% RSLogix 500 project 04_P9_ASHLEY_J.RSS, saved by version 8.30.00.16 %
PROJECT "UNTITLED"    % processor: Bul.1763 MicroLogix 1100 Series B %

PROGRAM FILES
  LAD 2 "MAIN"  3 rungs
  LAD 3 "MODE_CTRLS"  13 rungs
  LAD 4 "DATA_CTRL"  9 rungs

DATA FILES
  O0 OUTPUT  4 elements
  I1 INPUT  6 elements
  S2 STATUS  66 elements
  B3 BINARY  10 elements
  T4 TIMER  4 elements
  C5 COUNTER  1 elements
  R6 CONTROL  1 elements
  N7 INTEGER  4 elements
  F8 FLOAT  1 elements
  ST9 STRINGS  10 elements

LADDER 2 "MAIN"
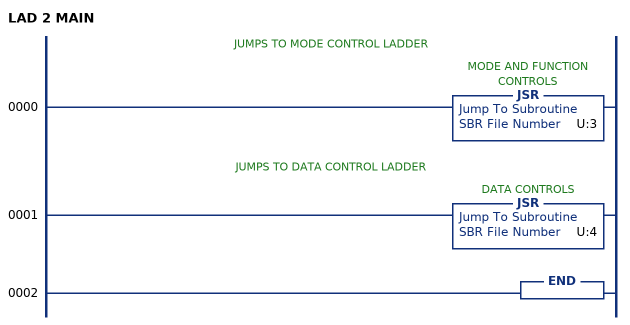
% Rung: 0 %
% JUMPS TO MODE CONTROL LADDER %
SOR JSR U:3 EOR
%   U:3  "MODE AND FUNCTION CONTROLS" %
% Rung: 1 %
% JUMPS TO DATA CONTROL LADDER %
SOR JSR U:4 EOR
%   U:4  "DATA CONTROLS" %
% Rung: 2 %
SOR END EOR

LADDER 3 "MODE_CTRLS"
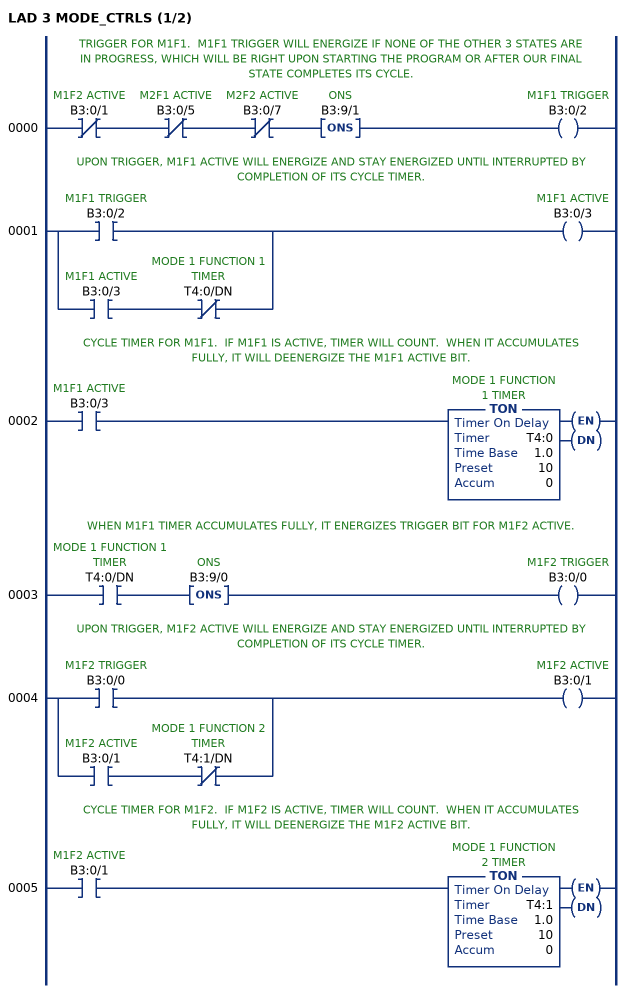
% Rung: 0 %
% TRIGGER FOR M1F1.  M1F1 TRIGGER WILL ENERGIZE IF NONE OF THE OTHER 3 STATES ARE IN PROGRESS, WHICH WILL BE RIGHT UPON STARTING THE PROGRAM OR AFTER OUR FINAL STATE COMPLETES ITS CYCLE. %
SOR XIO B3:0/1 XIO B3:0/5 XIO B3:0/7 ONS B3:9/1 OTE B3:0/2 EOR
%   B3:0/1  "M1F2 ACTIVE" %
%   B3:0/5  "M2F1 ACTIVE" %
%   B3:0/7  "M2F2 ACTIVE" %
%   B3:9/1  "ONS" %
%   B3:0/2  "M1F1 TRIGGER" %
% Rung: 1 %
% UPON TRIGGER, M1F1 ACTIVE WILL ENERGIZE AND STAY ENERGIZED UNTIL INTERRUPTED BY COMPLETION OF ITS CYCLE TIMER. %
SOR BST XIC B3:0/2 NXB XIC B3:0/3 XIO T4:0/DN BND OTE B3:0/3 EOR
%   B3:0/2  "M1F1 TRIGGER" %
%   B3:0/3  "M1F1 ACTIVE" %
%   T4:0  "MODE 1 FUNCTION 1 TIMER" %
% Rung: 2 %
% CYCLE TIMER FOR M1F1.  IF M1F1 IS ACTIVE, TIMER WILL COUNT.  WHEN IT ACCUMULATES FULLY, IT WILL DEENERGIZE THE M1F1 ACTIVE BIT. %
SOR XIC B3:0/3 TON T4:0 1.0 10 0 EOR
%   B3:0/3  "M1F1 ACTIVE" %
%   T4:0  "MODE 1 FUNCTION 1 TIMER" %
% Rung: 3 %
% WHEN M1F1 TIMER ACCUMULATES FULLY, IT ENERGIZES TRIGGER BIT FOR M1F2 ACTIVE. %
SOR XIC T4:0/DN ONS B3:9/0 OTE B3:0/0 EOR
%   T4:0  "MODE 1 FUNCTION 1 TIMER" %
%   B3:9/0  "ONS" %
%   B3:0/0  "M1F2 TRIGGER" %
% Rung: 4 %
% UPON TRIGGER, M1F2 ACTIVE WILL ENERGIZE AND STAY ENERGIZED UNTIL INTERRUPTED BY COMPLETION OF ITS CYCLE TIMER. %
SOR BST XIC B3:0/0 NXB XIC B3:0/1 XIO T4:1/DN BND OTE B3:0/1 EOR
%   B3:0/0  "M1F2 TRIGGER" %
%   B3:0/1  "M1F2 ACTIVE" %
%   T4:1  "MODE 1 FUNCTION 2 TIMER" %
% Rung: 5 %
% CYCLE TIMER FOR M1F2.  IF M1F2 IS ACTIVE, TIMER WILL COUNT.  WHEN IT ACCUMULATES FULLY, IT WILL DEENERGIZE THE M1F2 ACTIVE BIT. %
SOR XIC B3:0/1 TON T4:1 1.0 10 0 EOR
%   B3:0/1  "M1F2 ACTIVE" %
%   T4:1  "MODE 1 FUNCTION 2 TIMER" %

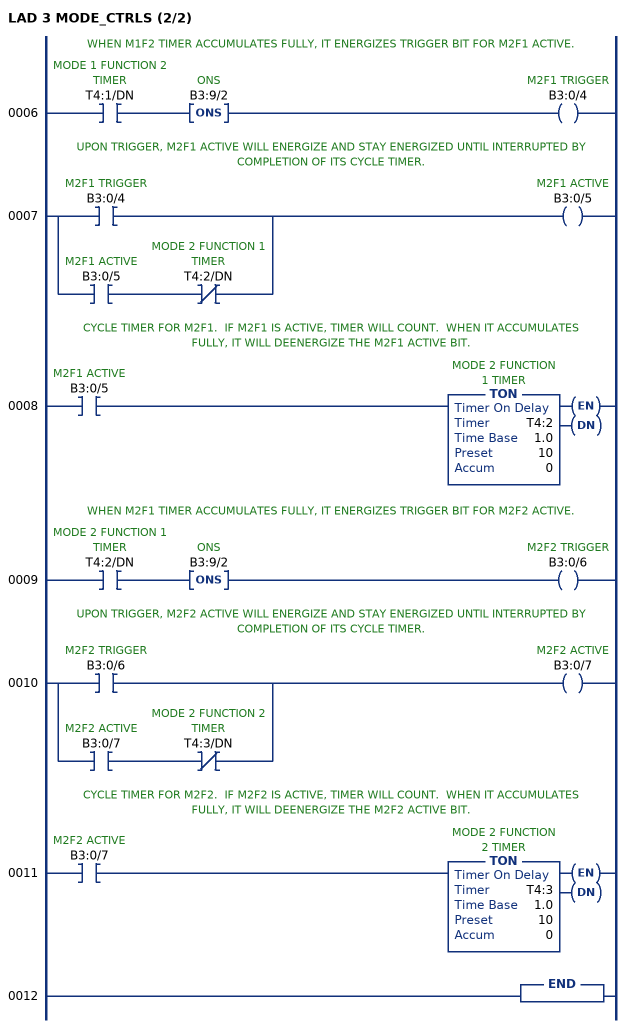
% Rung: 6 %
% WHEN M1F2 TIMER ACCUMULATES FULLY, IT ENERGIZES TRIGGER BIT FOR M2F1 ACTIVE. %
SOR XIC T4:1/DN ONS B3:9/2 OTE B3:0/4 EOR
%   T4:1  "MODE 1 FUNCTION 2 TIMER" %
%   B3:9/2  "ONS" %
%   B3:0/4  "M2F1 TRIGGER" %
% Rung: 7 %
% UPON TRIGGER, M2F1 ACTIVE WILL ENERGIZE AND STAY ENERGIZED UNTIL INTERRUPTED BY COMPLETION OF ITS CYCLE TIMER. %
SOR BST XIC B3:0/4 NXB XIC B3:0/5 XIO T4:2/DN BND OTE B3:0/5 EOR
%   B3:0/4  "M2F1 TRIGGER" %
%   B3:0/5  "M2F1 ACTIVE" %
%   T4:2  "MODE 2 FUNCTION 1 TIMER" %
% Rung: 8 %
% CYCLE TIMER FOR M2F1.  IF M2F1 IS ACTIVE, TIMER WILL COUNT.  WHEN IT ACCUMULATES FULLY, IT WILL DEENERGIZE THE M2F1 ACTIVE BIT. %
SOR XIC B3:0/5 TON T4:2 1.0 10 0 EOR
%   B3:0/5  "M2F1 ACTIVE" %
%   T4:2  "MODE 2 FUNCTION 1 TIMER" %
% Rung: 9 %
% WHEN M2F1 TIMER ACCUMULATES FULLY, IT ENERGIZES TRIGGER BIT FOR M2F2 ACTIVE. %
SOR XIC T4:2/DN ONS B3:9/2 OTE B3:0/6 EOR
%   T4:2  "MODE 2 FUNCTION 1 TIMER" %
%   B3:9/2  "ONS" %
%   B3:0/6  "M2F2 TRIGGER" %
% Rung: 10 %
% UPON TRIGGER, M2F2 ACTIVE WILL ENERGIZE AND STAY ENERGIZED UNTIL INTERRUPTED BY COMPLETION OF ITS CYCLE TIMER. %
SOR BST XIC B3:0/6 NXB XIC B3:0/7 XIO T4:3/DN BND OTE B3:0/7 EOR
%   B3:0/6  "M2F2 TRIGGER" %
%   B3:0/7  "M2F2 ACTIVE" %
%   T4:3  "MODE 2 FUNCTION 2 TIMER" %
% Rung: 11 %
% CYCLE TIMER FOR M2F2.  IF M2F2 IS ACTIVE, TIMER WILL COUNT.  WHEN IT ACCUMULATES FULLY, IT WILL DEENERGIZE THE M2F2 ACTIVE BIT. %
SOR XIC B3:0/7 TON T4:3 1.0 10 0 EOR
%   B3:0/7  "M2F2 ACTIVE" %
%   T4:3  "MODE 2 FUNCTION 2 TIMER" %
% Rung: 12 %
SOR END EOR

LADDER 4 "DATA_CTRL"
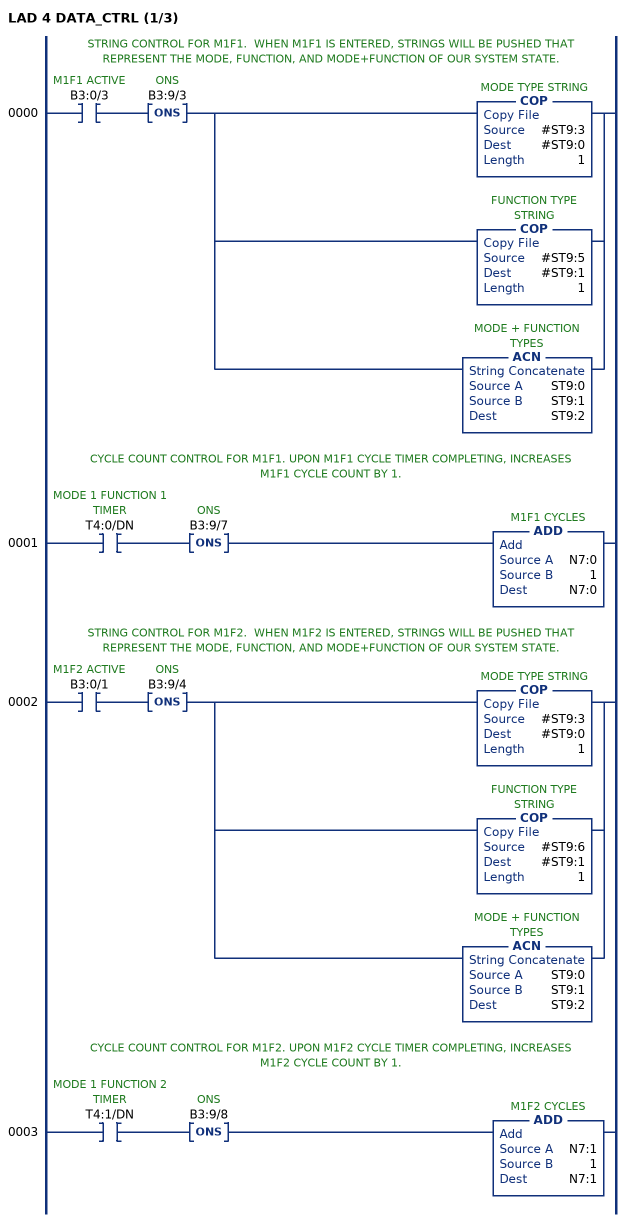
% Rung: 0 %
% STRING CONTROL FOR M1F1.  WHEN M1F1 IS ENTERED, STRINGS WILL BE PUSHED THAT REPRESENT THE MODE, FUNCTION, AND MODE+FUNCTION OF OUR SYSTEM STATE. %
SOR XIC B3:0/3 ONS B3:9/3 BST COP #ST9:3 #ST9:0 1 NXB COP #ST9:5 #ST9:1 1 NXB ACN ST9:0 ST9:1 ST9:2 BND EOR
%   B3:0/3  "M1F1 ACTIVE" %
%   B3:9/3  "ONS" %
%   ST9:3  "MODE_1 STRING" %
%   ST9:0  "MODE TYPE STRING" %
%   ST9:5  "FUNCTION_1 STRING" %
%   ST9:1  "FUNCTION TYPE STRING" %
%   ST9:2  "MODE + FUNCTION TYPES" %
% Rung: 1 %
% CYCLE COUNT CONTROL FOR M1F1. UPON M1F1 CYCLE TIMER COMPLETING, INCREASES M1F1 CYCLE COUNT BY 1. %
SOR XIC T4:0/DN ONS B3:9/7 ADD N7:0 1 N7:0 EOR
%   T4:0  "MODE 1 FUNCTION 1 TIMER" %
%   B3:9/7  "ONS" %
%   N7:0  "M1F1 CYCLES" %
% Rung: 2 %
% STRING CONTROL FOR M1F2.  WHEN M1F2 IS ENTERED, STRINGS WILL BE PUSHED THAT REPRESENT THE MODE, FUNCTION, AND MODE+FUNCTION OF OUR SYSTEM STATE. %
SOR XIC B3:0/1 ONS B3:9/4 BST COP #ST9:3 #ST9:0 1 NXB COP #ST9:6 #ST9:1 1 NXB ACN ST9:0 ST9:1 ST9:2 BND EOR
%   B3:0/1  "M1F2 ACTIVE" %
%   B3:9/4  "ONS" %
%   ST9:3  "MODE_1 STRING" %
%   ST9:0  "MODE TYPE STRING" %
%   ST9:6  "FUNCTION_2 STRING" %
%   ST9:1  "FUNCTION TYPE STRING" %
%   ST9:2  "MODE + FUNCTION TYPES" %
% Rung: 3 %
% CYCLE COUNT CONTROL FOR M1F2. UPON M1F2 CYCLE TIMER COMPLETING, INCREASES M1F2 CYCLE COUNT BY 1. %
SOR XIC T4:1/DN ONS B3:9/8 ADD N7:1 1 N7:1 EOR
%   T4:1  "MODE 1 FUNCTION 2 TIMER" %
%   B3:9/8  "ONS" %
%   N7:1  "M1F2 CYCLES" %

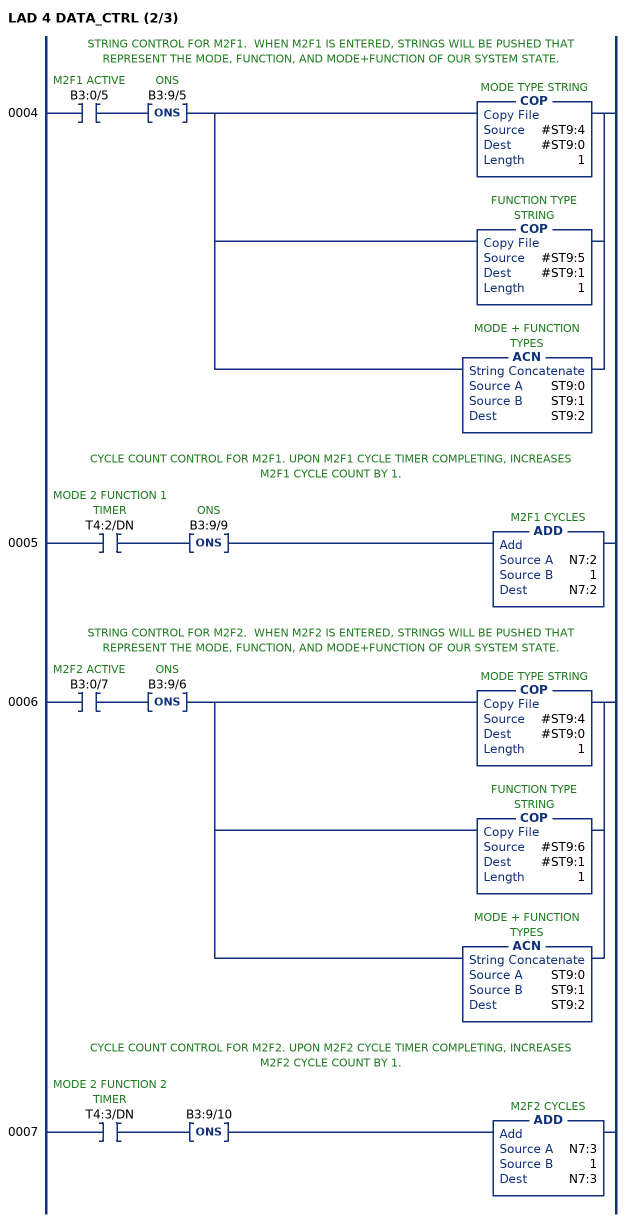
% Rung: 4 %
% STRING CONTROL FOR M2F1.  WHEN M2F1 IS ENTERED, STRINGS WILL BE PUSHED THAT REPRESENT THE MODE, FUNCTION, AND MODE+FUNCTION OF OUR SYSTEM STATE. %
SOR XIC B3:0/5 ONS B3:9/5 BST COP #ST9:4 #ST9:0 1 NXB COP #ST9:5 #ST9:1 1 NXB ACN ST9:0 ST9:1 ST9:2 BND EOR
%   B3:0/5  "M2F1 ACTIVE" %
%   B3:9/5  "ONS" %
%   ST9:4  "MODE_2 STRING" %
%   ST9:0  "MODE TYPE STRING" %
%   ST9:5  "FUNCTION_1 STRING" %
%   ST9:1  "FUNCTION TYPE STRING" %
%   ST9:2  "MODE + FUNCTION TYPES" %
% Rung: 5 %
% CYCLE COUNT CONTROL FOR M2F1. UPON M2F1 CYCLE TIMER COMPLETING, INCREASES M2F1 CYCLE COUNT BY 1. %
SOR XIC T4:2/DN ONS B3:9/9 ADD N7:2 1 N7:2 EOR
%   T4:2  "MODE 2 FUNCTION 1 TIMER" %
%   B3:9/9  "ONS" %
%   N7:2  "M2F1 CYCLES" %
% Rung: 6 %
% STRING CONTROL FOR M2F2.  WHEN M2F2 IS ENTERED, STRINGS WILL BE PUSHED THAT REPRESENT THE MODE, FUNCTION, AND MODE+FUNCTION OF OUR SYSTEM STATE. %
SOR XIC B3:0/7 ONS B3:9/6 BST COP #ST9:4 #ST9:0 1 NXB COP #ST9:6 #ST9:1 1 NXB ACN ST9:0 ST9:1 ST9:2 BND EOR
%   B3:0/7  "M2F2 ACTIVE" %
%   B3:9/6  "ONS" %
%   ST9:4  "MODE_2 STRING" %
%   ST9:0  "MODE TYPE STRING" %
%   ST9:6  "FUNCTION_2 STRING" %
%   ST9:1  "FUNCTION TYPE STRING" %
%   ST9:2  "MODE + FUNCTION TYPES" %
% Rung: 7 %
% CYCLE COUNT CONTROL FOR M2F2. UPON M2F2 CYCLE TIMER COMPLETING, INCREASES M2F2 CYCLE COUNT BY 1. %
SOR XIC T4:3/DN ONS B3:9/10 ADD N7:3 1 N7:3 EOR
%   T4:3  "MODE 2 FUNCTION 2 TIMER" %
%   N7:3  "M2F2 CYCLES" %

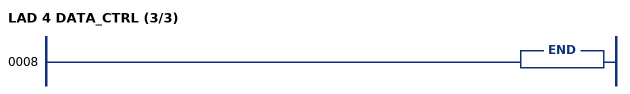
% Rung: 8 %
SOR END EOR

DATA TABLE (non-zero values as saved)
DATA T4
% .PRE .ACC %
% T4:0 % 10 0
% T4:1 % 10 0
% T4:2 % 10 0
% T4:3 % 10 0
DATA ST9
% ST9:3 % "MODE_1 "
% ST9:4 % "MODE_2 "
% ST9:5 % "FUNCTION_1"
% ST9:6 % "FUNCTION_2"
